// LS Electric XG5000 project: 동남82
// PLC NewPLC
// module base 0 slot 0: 입출력 모듈:XBC-DN/DP14E (DC 24V 입력 8점, 트랜지스터 출력 6점)

PROGRAM NewProgram (task: 스캔 프로그램)

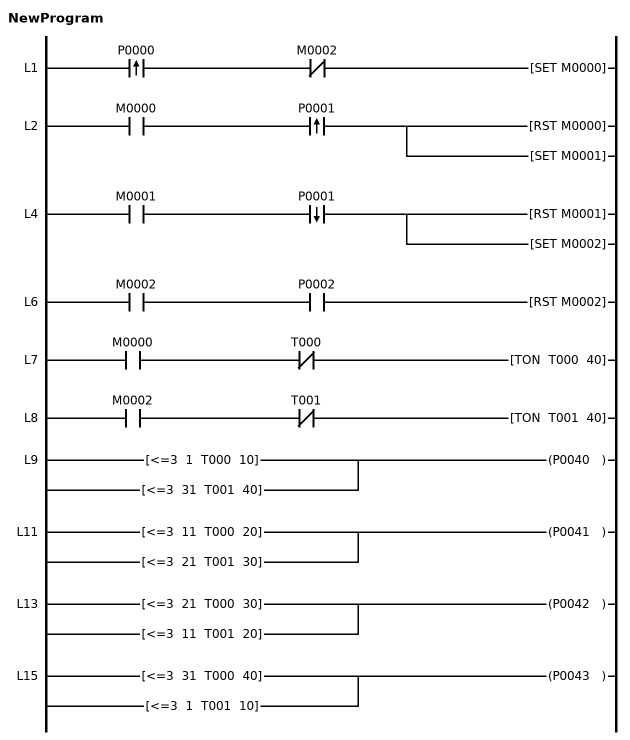
; L1
LOADP     P0000
AND NOT   M0002
SET       M0000
; L2
LOAD      M0000
ANDP      P0001
RST       M0000
SET       M0001
; L4
LOAD      M0001
ANDN      P0001
RST       M0001
SET       M0002
; L6
LOAD      M0002
AND       P0002
RST       M0002
; L7
LOAD      M0000
AND NOT   T000
TON       T000 40
; L8
LOAD      M0002
AND NOT   T001
TON       T001 40
; L9
LOAD<=3   1 T000 10
OR<=3     31 T001 40
OUT       P0040
; L11
LOAD<=3   11 T000 20
OR<=3     21 T001 30
OUT       P0041
; L13
LOAD<=3   21 T000 30
OR<=3     11 T001 20
OUT       P0042
; L15
LOAD<=3   31 T000 40
OR<=3     1 T001 10
OUT       P0043